Staubli VAL3: motionWorker.pgx

program motionWorker()
begin

  while true
    wait(motionQueued)
    motionQueued = false

    if motionType == 0
      logMsg("[MOTION] Linear move")
      movel(target, selectedTool, moveConfig)

    elseIf motionType == 1
      logMsg("[MOTION] Direct move")
      movej(target, selectedTool, moveConfig)

    elseIf motionType == 2
      logMsg("[MOTION] Joint move")
      movej(pose, selectedTool, moveConfig)

    elseIf motionType == 3
      logMsg("[MOTION] Circular move")
      movec(intermediate, target, selectedTool, moveConfig)
    endIf

  endWhile
end
